Fanuc KAREL source: NC0072.KL

-- PROVISIONAL review KL for V1013-1; original PC SHA256 6bb5e675d689680fce8d14dd052e9c91cf3c6f9823a512edb3392a26699f1ab2
-- Incomplete behavior may be omitted. Consult companion uncertainty JSON. Do not deploy.
PROGRAM NC0072
%NOLOCKGROUP
-- UNRESOLVED_LOCAL_POOL 1 cells at code offset 3; source declarations unknown
-- DIRECT_LOCAL_WORD_ACCESS alone does not prove INTEGER, REAL, or BOOLEAN
BEGIN
  -- UNRESOLVED_PC offsets 0-8; opcodes 2B,2C,7B
  -- UNRESOLVED_PC offsets 13-20; opcodes 9D,23
  -- UNRESOLVED_PC offsets 25-42; opcodes 21,2E,59,79
  -- UNRESOLVED_PC offsets 47-61; opcodes 21,9D,52,23
  -- UNRESOLVED_PC offsets 66-71; opcodes 7A
  -- UNRESOLVED_PC offsets 76-80; opcodes 7F
  -- UNRESOLVED_PC offsets 85-89; opcodes 27,AA
  -- UNRESOLVED_PC offsets 94-98; opcodes 7F
END NC0072
